FUNCTION_BLOCK FB_MasterSlaveCheckDetect
VAR_INPUT
END_VAR
VAR_OUTPUT
END_VAR
VAR
	m_salveCheckCounts :INT :=0;
	m_salveCheckThres :INT :=10;
END_VAR

// check if instrument is on
METHOD run : BOOL
VAR_INPUT
	IOValue :BOOL;
END_VAR

IF IOValue = TRUE  THEN
	m_salveCheckCounts := MIN( m_salveCheckCounts +1,m_salveCheckThres);
ELSIF IOValue = FALSE  THEN
	m_salveCheckCounts :=0;
END_IF
run := m_salveCheckCounts >= m_salveCheckThres;
END_METHOD

END_FUNCTION_BLOCK

(* stored: Version 1.1.0.1, ProductVersion 3.1.4024.11
   POU FB_MasterSlaveCheckDetect: Id {2fc52dc6-aea9-4f7f-9696-53f309e4debb}, SpecialFunc None
   Method run: Id {c4c42e8a-47e4-4b2e-af21-67d5fd4387a7} *)
